TYPE
    TcoControlledZone_Config :
    STRUCT
        MaxControledUnits : USINT := 12;
        MaxControlButtons : USINT := 4;
        MaxKeyMode : USINT := 4;
        MaxKeyNormalService : USINT := 4;
        DoorsLocked : TIME := T#1S;
    END_STRUCT
END_TYPE

(* stored: Version 1.1.0.1
   DUT TcoControlledZone_Config: Id {1a75dab5-4912-4cfc-b5a7-3092971d60ad} *)
